{attribute 'c++_compatible'}
{attribute 'external_name' := 'EncoderTouchProbeRef_GUID_799525EC_5EF1_E852_EDA3_1BA0CDBD1FD9'}
{attribute 'TcIecLibraryType'}
{attribute 'no_explicit_call' :='do not call this POU directly'}
{attribute 'no_assign_warning'}
(* TouchProbeRef for Encoder Touch Probe. *)
FUNCTION_BLOCK EncoderTouchProbeRef
VAR
END_VAR
VAR_INPUT
	(* Settings for incremental encoder touch probe source selection. *)
	{attribute 'GUID' := '150DF3A8-F3D9-498D-A6F5-12073AD04A71'}
	{attribute 'Namespace' := 'Tc3_Mc3Ptp'}
	IncrementalEncoderSettings : IncrementalEncoderTouchProbeSettings;
END_VAR
VAR
	 {attribute 'hide'}
	_reserved1 : UDINT;
END_VAR
VAR_OUTPUT
	(* Connect to MC_TouchProbe/MC_AbortTrigger TriggerInput *)
	{attribute 'GUID' := 'CC3262A1-A7A1-46D3-802E-9117404E77E7'}
	{attribute 'Namespace' := 'Tc3_Mc3Ptp'}
	Trigger : TRIGGER_REF;
END_VAR
VAR
	 {attribute 'hide'}
	_reserved2 : ARRAY [1..8] OF USINT;
END_VAR

{attribute 'TcTypeSystem'}

(* Internal method *)
{attribute 'hide'}
METHOD FB_init : BOOL
VAR_INPUT
	(*  if TRUE, the retain variables are initialized (warm start / cold start) *)
	bInitRetains : BOOL;
	(*  if TRUE, the instance afterwards gets moved into the copy code (online change) *)
	bInCopyCode : BOOL;
END_VAR
END_METHOD

{attribute 'TcTypeSystem'}

(* Internal method *)
{attribute 'hide'}
METHOD FB_reinit : BOOL
END_METHOD

{attribute 'TcTypeSystem'}

(* Internal method *)
{attribute 'hide'}
METHOD FB_exit : BOOL
VAR_INPUT
	(*  if TRUE, the exit method is called for exiting an instance that is copied afterwards (online change). *)
	bInCopyCode : BOOL;
END_VAR
END_METHOD

END_FUNCTION_BLOCK

// TouchProbe/TimestampTouchProbeRef

{attribute 'c++_compatible'}
{attribute 'external_name' := 'TimestampTouchProbeRef_GUID_B6855340_6F16_E41B_E060_D5170EE631A7'}
{attribute 'TcIecLibraryType'}
{attribute 'no_explicit_call' :='do not call this POU directly'}
{attribute 'no_assign_warning'}
(* TouchProbeRef for Timestamp Touch Probes. *)
FUNCTION_BLOCK TimestampTouchProbeRef
VAR
END_VAR
VAR_INPUT
	(* Link to Axis Touch Probe Object -> Oid. *)
	{attribute 'GUID' := '18071995-0000-0000-0000-00000000000F'}
	Oid AT %I* : GLOBAL.OTCID;
END_VAR
VAR
	 {attribute 'hide'}
	_reserved1 : UDINT;
END_VAR
VAR_OUTPUT
	(* Connect to MC_Touchprobe/MC_AbortTrigger TriggerInput *)
	{attribute 'GUID' := 'CC3262A1-A7A1-46D3-802E-9117404E77E7'}
	{attribute 'Namespace' := 'Tc3_Mc3Ptp'}
	Trigger : TRIGGER_REF;
END_VAR

{attribute 'TcTypeSystem'}

(* Internal method *)
{attribute 'hide'}
METHOD FB_init : BOOL
VAR_INPUT
	(*  if TRUE, the retain variables are initialized (warm start / cold start) *)
	bInitRetains : BOOL;
	(*  if TRUE, the instance afterwards gets moved into the copy code (online change) *)
	bInCopyCode : BOOL;
END_VAR
END_METHOD

{attribute 'TcTypeSystem'}

(* Internal method *)
{attribute 'hide'}
METHOD FB_reinit : BOOL
END_METHOD

{attribute 'TcTypeSystem'}

(* Internal method *)
{attribute 'hide'}
METHOD FB_exit : BOOL
VAR_INPUT
	(*  if TRUE, the exit method is called for exiting an instance that is copied afterwards (online change). *)
	bInCopyCode : BOOL;
END_VAR
END_METHOD

END_FUNCTION_BLOCK

// TouchProbe/FixedStopTouchProbeRef

{attribute 'c++_compatible'}
{attribute 'external_name' := 'FixedStopTouchProbeRef_GUID_6C680BDF_D95B_EB97_DB3C_C590086A417A'}
{attribute 'TcIecLibraryType'}
{attribute 'no_explicit_call' :='do not call this POU directly'}
{attribute 'no_assign_warning'}
(* TouchProbeRef for Fixed Stop Detection. *)
FUNCTION_BLOCK FixedStopTouchProbeRef
VAR
END_VAR
VAR_INPUT
	(* Link to Axis Touch Probe Object -> Oid. *)
	{attribute 'GUID' := '18071995-0000-0000-0000-00000000000F'}
	Oid AT %I* : GLOBAL.OTCID;
END_VAR
VAR
	 {attribute 'hide'}
	_reserved1 : UDINT;
END_VAR
VAR_INPUT
	(* Settings for Fixed Stop Detection *)
	{attribute 'GUID' := 'CB5E9FDE-923C-4F7A-BCB2-279EC887599F'}
	{attribute 'Namespace' := 'Tc3_Mc3Ptp'}
	Settings : FixedStopTouchProbeSettings;
END_VAR
VAR_OUTPUT
	(* Connect to MC_Touchprobe/MC_AbortTrigger TriggerInput *)
	{attribute 'GUID' := 'CC3262A1-A7A1-46D3-802E-9117404E77E7'}
	{attribute 'Namespace' := 'Tc3_Mc3Ptp'}
	Trigger : TRIGGER_REF;
END_VAR

{attribute 'TcTypeSystem'}

(* Internal method *)
{attribute 'hide'}
METHOD FB_init : BOOL
VAR_INPUT
	(*  if TRUE, the retain variables are initialized (warm start / cold start) *)
	bInitRetains : BOOL;
	(*  if TRUE, the instance afterwards gets moved into the copy code (online change) *)
	bInCopyCode : BOOL;
END_VAR
END_METHOD

{attribute 'TcTypeSystem'}

(* Internal method *)
{attribute 'hide'}
METHOD FB_reinit : BOOL
END_METHOD

{attribute 'TcTypeSystem'}

(* Internal method *)
{attribute 'hide'}
METHOD FB_exit : BOOL
VAR_INPUT
	(*  if TRUE, the exit method is called for exiting an instance that is copied afterwards (online change). *)
	bInCopyCode : BOOL;
END_VAR
END_METHOD

END_FUNCTION_BLOCK

// Load Control/MC_LoadControl

{attribute 'c++_compatible'}
{attribute 'external_name' := 'MC_LoadControl_GUID_66886162_A3C4_E2E4_F654_8D3CE3C1FC4A'}
{attribute 'TcIecLibraryType'}
{attribute 'hide_all_locals'}
(* 
	This function block continuously exerts a torque, force or pressure of the specified value. <br/>
	Positive torque, force and differential pressure is in the positive direction of velocity, pressure is
	physically unsigned. LoadUnit must match the unit of the value measured by the corresponding sensor.
	 *)
FUNCTION_BLOCK MC_LoadControl
VAR_IN_OUT
	(* Reference to the axis *)
	{attribute 'GUID' := '931209B0-6FAC-E9BE-F824-23CE2FAA5732'}
	{attribute 'Namespace' := 'Tc3_Mc3Ptp'}
	Axis : AXIS_REF;
END_VAR
VAR_INPUT
	(* Start the motion at rising edge. *)
	Execute : BOOL;
END_VAR
VAR
	 {attribute 'hide'}
	_reserved1 : ARRAY [1..7] OF USINT;
END_VAR
VAR_INPUT
	(* Commanded load value ([LoadUnit]). It is approached using a defined ramp (LoadRamp). *)
	Load : LREAL := STRING_TO_LREAL('#Invalid');
	(* Maximum load derivative ([LoadUnit/s], positive) *)
	LoadRamp : LREAL := STRING_TO_LREAL('#Invalid');
	(* Maximum load ramp derivative ([LoadUnit/s^2], positive). It can be left as 'Ignore' if no ramp derivative limit is desired. *)
	LoadRampDerivative : LREAL := STRING_TO_LREAL('#Ignore');
	(* Chronological sequence of the command *)
	{attribute 'Namespace' := 'Tc3_Mc3Base'}
	BufferMode : Tc3_Mc3Base.EBufferMode := Tc3_Mc3Base.EBufferMode.Aborting;
END_VAR
VAR_OUTPUT
	(* Commanded load value reached *)
	InLoad : BOOL;
	(* Function block is not finished and new output values are to be expected. *)
	Busy : BOOL;
	(* Function block has active control on the axis. *)
	Active : BOOL;
	(* Command is aborted by another command. *)
	CommandAborted : BOOL;
	(* Error occurred within function block. *)
	Error : BOOL;
END_VAR
VAR
	 {attribute 'hide'}
	_reserved2 : USINT;
END_VAR
VAR_OUTPUT
	(* Error identifier *)
	ErrorId : UDINT;
END_VAR
VAR
	 {attribute 'hide'}
	_reserved3 : UINT_0_32;
	 {attribute 'hide'}
	_reserved4 : ARRAY [1..28] OF UINT_8_16;
	 {attribute 'hide'}
	_reserved5 : ARRAY [1..32] OF USINT;
END_VAR

{attribute 'TcTypeSystem'}

(* Internal method *)
{attribute 'hide'}
METHOD FB_init : BOOL
VAR_INPUT
	(*  if TRUE, the retain variables are initialized (warm start / cold start) *)
	bInitRetains : BOOL;
	(*  if TRUE, the instance afterwards gets moved into the copy code (online change) *)
	bInCopyCode : BOOL;
END_VAR
END_METHOD

{attribute 'TcTypeSystem'}

(* Internal method *)
{attribute 'hide'}
METHOD FB_exit : BOOL
VAR_INPUT
	(*  if TRUE, the exit method is called for exiting an instance that is copied afterwards (online change). *)
	bInCopyCode : BOOL;
END_VAR
END_METHOD

END_FUNCTION_BLOCK

// Administrative/Status/MC_ReadActualPosition

{attribute 'c++_compatible'}
{attribute 'external_name' := 'MC_ReadActualPosition_GUID_2E787536_22C6_ED03_C885_6ED50CC1B12A'}
{attribute 'TcIecLibraryType'}
{attribute 'hide_all_locals'}
(* 
		This function block reads the current axis actual position.<br/>
		In case of an invalid actual position value, the Position output is set to 0 and the Valid output is set to FALSE.
	 *)
FUNCTION_BLOCK MC_ReadActualPosition
VAR_IN_OUT
	(* Reference to the axis *)
	{attribute 'GUID' := '931209B0-6FAC-E9BE-F824-23CE2FAA5732'}
	{attribute 'Namespace' := 'Tc3_Mc3Ptp'}
	Axis : AXIS_REF;
END_VAR
VAR_INPUT
	(* Read the actual position continuously while Enable = TRUE. *)
	Enable : BOOL;
END_VAR
VAR_OUTPUT
	(* Valid output available at function block *)
	Valid : BOOL;
	(* Function block is not finished and new output values are to be expected. *)
	Busy : BOOL;
	(* Error occurred within function block. *)
	Error : BOOL;
	(* Error identifier *)
	ErrorId : UDINT;
	(* Actual position ([PosUnit]) *)
	Position : LREAL;
END_VAR

{attribute 'TcTypeSystem'}

(* Internal method *)
{attribute 'hide'}
METHOD FB_init : BOOL
VAR_INPUT
	(*  if TRUE, the retain variables are initialized (warm start / cold start) *)
	bInitRetains : BOOL;
	(*  if TRUE, the instance afterwards gets moved into the copy code (online change) *)
	bInCopyCode : BOOL;
END_VAR
END_METHOD

{attribute 'TcTypeSystem'}

(* Internal method *)
{attribute 'hide'}
METHOD FB_exit : BOOL
VAR_INPUT
	(*  if TRUE, the exit method is called for exiting an instance that is copied afterwards (online change). *)
	bInCopyCode : BOOL;
END_VAR
END_METHOD

END_FUNCTION_BLOCK

// Administrative/Status/MC_ReadActualTorque

{attribute 'c++_compatible'}
{attribute 'external_name' := 'MC_ReadActualTorque_GUID_AD684BB3_AFE8_E183_D73B_36C41C0C538D'}
{attribute 'TcIecLibraryType'}
{attribute 'hide_all_locals'}
(* 
		This function block reads the current axis actual torque.<br/>
		In case of an invalid actual torque value, the Torque output is set to 0 and the Valid output is set to FALSE.
	 *)
FUNCTION_BLOCK MC_ReadActualTorque
VAR_IN_OUT
	(* Reference to the axis *)
	{attribute 'GUID' := '931209B0-6FAC-E9BE-F824-23CE2FAA5732'}
	{attribute 'Namespace' := 'Tc3_Mc3Ptp'}
	Axis : AXIS_REF;
END_VAR
VAR_INPUT
	(* Read the actual torque continuously while Enable = TRUE. *)
	Enable : BOOL;
END_VAR
VAR_OUTPUT
	(* Valid output available at function block *)
	Valid : BOOL;
	(* Function block is not finished and new output values are to be expected. *)
	Busy : BOOL;
	(* Error occurred within function block. *)
	Error : BOOL;
	(* Error identifier *)
	ErrorId : UDINT;
	(* Actual torque ([TorqueUnit]) *)
	Torque : LREAL;
END_VAR

{attribute 'TcTypeSystem'}

(* Internal method *)
{attribute 'hide'}
METHOD FB_init : BOOL
VAR_INPUT
	(*  if TRUE, the retain variables are initialized (warm start / cold start) *)
	bInitRetains : BOOL;
	(*  if TRUE, the instance afterwards gets moved into the copy code (online change) *)
	bInCopyCode : BOOL;
END_VAR
END_METHOD

{attribute 'TcTypeSystem'}

(* Internal method *)
{attribute 'hide'}
METHOD FB_exit : BOOL
VAR_INPUT
	(*  if TRUE, the exit method is called for exiting an instance that is copied afterwards (online change). *)
	bInCopyCode : BOOL;
END_VAR
END_METHOD

END_FUNCTION_BLOCK

// Administrative/Status/MC_ReadActualVelocity

{attribute 'c++_compatible'}
{attribute 'external_name' := 'MC_ReadActualVelocity_GUID_DD1D8D4C_516C_E0E0_F57B_12AC9CA1B220'}
{attribute 'TcIecLibraryType'}
{attribute 'hide_all_locals'}
(* 
		This function block reads the current axis actual velocity.<br/>
		In case of an invalid actual velocity value, the Velocity output is set to 0 and the Valid output is set to FALSE.
	 *)
FUNCTION_BLOCK MC_ReadActualVelocity
VAR_IN_OUT
	(* Reference to the axis *)
	{attribute 'GUID' := '931209B0-6FAC-E9BE-F824-23CE2FAA5732'}
	{attribute 'Namespace' := 'Tc3_Mc3Ptp'}
	Axis : AXIS_REF;
END_VAR
VAR_INPUT
	(* Read the actual velocity continuously while Enable = TRUE. *)
	Enable : BOOL;
END_VAR
VAR_OUTPUT
	(* Valid output available at function block *)
	Valid : BOOL;
	(* Function block is not finished and new output values are to be expected. *)
	Busy : BOOL;
	(* Error occurred within function block. *)
	Error : BOOL;
	(* Error identifier *)
	ErrorId : UDINT;
	(* Actual velocity ([PosUnit]/s) *)
	Velocity : LREAL;
END_VAR

{attribute 'TcTypeSystem'}

(* Internal method *)
{attribute 'hide'}
METHOD FB_init : BOOL
VAR_INPUT
	(*  if TRUE, the retain variables are initialized (warm start / cold start) *)
	bInitRetains : BOOL;
	(*  if TRUE, the instance afterwards gets moved into the copy code (online change) *)
	bInCopyCode : BOOL;
END_VAR
END_METHOD

{attribute 'TcTypeSystem'}

(* Internal method *)
{attribute 'hide'}
METHOD FB_exit : BOOL
VAR_INPUT
	(*  if TRUE, the exit method is called for exiting an instance that is copied afterwards (online change). *)
	bInCopyCode : BOOL;
END_VAR
END_METHOD

END_FUNCTION_BLOCK

// Administrative/Status/MC_ReadAxisError

{attribute 'c++_compatible'}
{attribute 'external_name' := 'MC_ReadAxisError_GUID_161A2F0B_30EC_E528_DEE0_A4EC734D4B38'}
{attribute 'TcIecLibraryType'}
{attribute 'hide_all_locals'}
(* 
		This function block reads the current axis error identifier.
	 *)
FUNCTION_BLOCK MC_ReadAxisError
VAR_IN_OUT
	(* Reference to the axis *)
	{attribute 'GUID' := '931209B0-6FAC-E9BE-F824-23CE2FAA5732'}
	{attribute 'Namespace' := 'Tc3_Mc3Ptp'}
	Axis : AXIS_REF;
END_VAR
VAR_INPUT
	(* Read the axis error identifier continuously while Enable = TRUE. *)
	Enable : BOOL;
END_VAR
VAR_OUTPUT
	(* Valid output available at function block *)
	Valid : BOOL;
	(* Function block is not finished and new output values are to be expected. *)
	Busy : BOOL;
	(* Error occurred within function block. *)
	Error : BOOL;
	(* Error identifier *)
	ErrorId : UDINT;
	(* Axis error identifier *)
	AxisErrorId : UDINT;
END_VAR
VAR
	 {attribute 'hide'}
	_reserved1 : UINT_0_32;
END_VAR

{attribute 'TcTypeSystem'}

(* Internal method *)
{attribute 'hide'}
METHOD FB_init : BOOL
VAR_INPUT
	(*  if TRUE, the retain variables are initialized (warm start / cold start) *)
	bInitRetains : BOOL;
	(*  if TRUE, the instance afterwards gets moved into the copy code (online change) *)
	bInCopyCode : BOOL;
END_VAR
END_METHOD

{attribute 'TcTypeSystem'}

(* Internal method *)
{attribute 'hide'}
METHOD FB_exit : BOOL
VAR_INPUT
	(*  if TRUE, the exit method is called for exiting an instance that is copied afterwards (online change). *)
	bInCopyCode : BOOL;
END_VAR
END_METHOD

END_FUNCTION_BLOCK

// Administrative/Status/MC_ReadStatus

{attribute 'c++_compatible'}
{attribute 'external_name' := 'MC_ReadStatus_GUID_BDF6D356_383A_E775_CF5E_17BC66992CB4'}
{attribute 'TcIecLibraryType'}
{attribute 'hide_all_locals'}
(* 
		This function block reads the current axis state.
	 *)
FUNCTION_BLOCK MC_ReadStatus
VAR_IN_OUT
	(* Reference to the axis *)
	{attribute 'GUID' := '931209B0-6FAC-E9BE-F824-23CE2FAA5732'}
	{attribute 'Namespace' := 'Tc3_Mc3Ptp'}
	Axis : AXIS_REF;
END_VAR
VAR_INPUT
	(* Read the axis state continuously while Enable = TRUE. *)
	Enable : BOOL;
END_VAR
VAR_OUTPUT
	(* Valid output available at function block *)
	Valid : BOOL;
	(* Function block is not finished and new output values are to be expected. *)
	Busy : BOOL;
	(* Error occurred within function block. *)
	Error : BOOL;
	(* Error identifier *)
	ErrorId : UDINT;
	(* Axis is in state ErrorStop. *)
	ErrorStop : BOOL;
	(* Axis is in state Disabled. *)
	Disabled : BOOL;
	(* Axis is in state Stopping. *)
	Stopping : BOOL;
	(* Axis is in state Homing. *)
	Homing : BOOL;
	(* Axis is in state Standstill. *)
	Standstill : BOOL;
	(* Axis is in state DiscreteMotion. *)
	DiscreteMotion : BOOL;
	(* Axis is in state ContinuousMotion. *)
	ContinuousMotion : BOOL;
	(* Axis is in state SynchronizedMotion. *)
	SynchronizedMotion : BOOL;
END_VAR

{attribute 'TcTypeSystem'}

(* Internal method *)
{attribute 'hide'}
METHOD FB_init : BOOL
VAR_INPUT
	(*  if TRUE, the retain variables are initialized (warm start / cold start) *)
	bInitRetains : BOOL;
	(*  if TRUE, the instance afterwards gets moved into the copy code (online change) *)
	bInCopyCode : BOOL;
END_VAR
END_METHOD

{attribute 'TcTypeSystem'}

(* Internal method *)
{attribute 'hide'}
METHOD FB_exit : BOOL
VAR_INPUT
	(*  if TRUE, the exit method is called for exiting an instance that is copied afterwards (online change). *)
	bInCopyCode : BOOL;
END_VAR
END_METHOD

END_FUNCTION_BLOCK

// Administrative/Parameter/MC_WriteHardwareParameter

{attribute 'c++_compatible'}
{attribute 'external_name' := 'MC_WriteHardwareParameter_GUID_4D6A3EB3_2727_E24A_E1EB_F69B71611CB4'}
{attribute 'TcIecLibraryType'}
{attribute 'hide_all_locals'}
(* 
		This function block allows to write parameters to the hardware drive asynchronously via ADS. It supports CoE and SoE drives.
	 *)
FUNCTION_BLOCK MC_WriteHardwareParameter
VAR_IN_OUT
	(* Reference to the axis *)
	{attribute 'GUID' := '931209B0-6FAC-E9BE-F824-23CE2FAA5732'}
	{attribute 'Namespace' := 'Tc3_Mc3Ptp'}
	Axis : AXIS_REF;
END_VAR
VAR_INPUT
	(* Rising edge triggers the write operation. *)
	Execute : BOOL;
END_VAR
VAR
	 {attribute 'hide'}
	_reserved1 : USINT;
END_VAR
VAR_INPUT
	(* CoE object index or SoE IDN *)
	Index : UINT := 0;
	(* CoE sub index or SoE element *)
	SubIndex : USINT := 0;
END_VAR
VAR
	 {attribute 'hide'}
	_reserved2 : ARRAY [1..3] OF USINT;
END_VAR
VAR_INPUT
	(* Contains the address of the data. *)
	{attribute 'GUID' := '18071995-0000-0000-0000-000000000018'}
	SourceAddress : GLOBAL.PVOID := 0;
	(* Contains the size of the data. *)
	DataSize : UDINT := 0;
END_VAR
VAR_OUTPUT
	(* Value is successfully sent to the target. *)
	Done : BOOL;
	(* Function block is not finished. *)
	Busy : BOOL;
	(* Function block is active. *)
	Active : BOOL;
	(* Error occurred within function block. *)
	Error : BOOL;
	(* Error identifier *)
	ErrorId : UDINT;
END_VAR
VAR
	 {attribute 'hide'}
	_reserved3 : UINT_0_32;
	 {attribute 'hide'}
	_reserved4 : ARRAY [1..32] OF UINT_8_16;
	 {attribute 'hide'}
	_reserved5 : ARRAY [1..32] OF USINT;
END_VAR

{attribute 'TcTypeSystem'}

(* Internal method *)
{attribute 'hide'}
METHOD FB_init : BOOL
VAR_INPUT
	(*  if TRUE, the retain variables are initialized (warm start / cold start) *)
	bInitRetains : BOOL;
	(*  if TRUE, the instance afterwards gets moved into the copy code (online change) *)
	bInCopyCode : BOOL;
END_VAR
END_METHOD

{attribute 'TcTypeSystem'}

(* Internal method *)
{attribute 'hide'}
METHOD FB_exit : BOOL
VAR_INPUT
	(*  if TRUE, the exit method is called for exiting an instance that is copied afterwards (online change). *)
	bInCopyCode : BOOL;
END_VAR
END_METHOD

END_FUNCTION_BLOCK

// Administrative/Parameter/MC_ReadHardwareParameter

{attribute 'c++_compatible'}
{attribute 'external_name' := 'MC_ReadHardwareParameter_GUID_DBC0D23F_EDB5_E904_FCD0_3F6DCE5C9980'}
{attribute 'TcIecLibraryType'}
{attribute 'hide_all_locals'}
(* 
		This function block allows to read parameters from the hardware drive asynchronously via ADS. The function block supports CoE and SoE drives.
	 *)
FUNCTION_BLOCK MC_ReadHardwareParameter
VAR_IN_OUT
	(* Reference to the axis *)
	{attribute 'GUID' := '931209B0-6FAC-E9BE-F824-23CE2FAA5732'}
	{attribute 'Namespace' := 'Tc3_Mc3Ptp'}
	Axis : AXIS_REF;
END_VAR
VAR_INPUT
	(* Trigger the command with rising edge. *)
	Execute : BOOL;
END_VAR
VAR
	 {attribute 'hide'}
	_reserved1 : USINT;
END_VAR
VAR_INPUT
	(* CoE object index or SoE IDN *)
	Index : UINT := 0;
	(* CoE sub index or SoE element *)
	SubIndex : USINT := 0;
END_VAR
VAR
	 {attribute 'hide'}
	_reserved2 : ARRAY [1..3] OF USINT;
END_VAR
VAR_INPUT
	(* Contains the address of the destination buffer. *)
	{attribute 'GUID' := '18071995-0000-0000-0000-000000000018'}
	DestinationAddress : GLOBAL.PVOID := 0;
	(* Contains the size of the destination buffer. *)
	DataSize : UDINT := 0;
END_VAR
VAR_OUTPUT
	(* Value is successfully read from the target. *)
	Done : BOOL;
	(* Function block is not finished. *)
	Busy : BOOL;
	(* Function block is active. *)
	Active : BOOL;
	(* Error occurred within function block. *)
	Error : BOOL;
	(* Error identifier *)
	ErrorId : UDINT;
END_VAR
VAR
	 {attribute 'hide'}
	_reserved3 : UINT_0_32;
	 {attribute 'hide'}
	_reserved4 : ARRAY [1..32] OF UINT_8_16;
	 {attribute 'hide'}
	_reserved5 : ARRAY [1..32] OF USINT;
END_VAR

{attribute 'TcTypeSystem'}

(* Internal method *)
{attribute 'hide'}
METHOD FB_init : BOOL
VAR_INPUT
	(*  if TRUE, the retain variables are initialized (warm start / cold start) *)
	bInitRetains : BOOL;
	(*  if TRUE, the instance afterwards gets moved into the copy code (online change) *)
	bInCopyCode : BOOL;
END_VAR
END_METHOD

{attribute 'TcTypeSystem'}

(* Internal method *)
{attribute 'hide'}
METHOD FB_exit : BOOL
VAR_INPUT
	(*  if TRUE, the exit method is called for exiting an instance that is copied afterwards (online change). *)
	bInCopyCode : BOOL;
END_VAR
END_METHOD

END_FUNCTION_BLOCK

// Administrative/Parameter/MC_ReadParameter

{attribute 'c++_compatible'}
{attribute 'pack_mode' := '1'}
{attribute 'external_name' := 'MC_ReadParameter_GUID_FFD552A7_9EB3_EE4D_D310_ABB0C47D1F25'}
{attribute 'TcIecLibraryType'}
{attribute 'hide_all_locals'}
(* 
		This function block reads a numeric (LREAL) parameter value from the axis.<br/>
		The command is typically processed synchronously.
	 *)
FUNCTION_BLOCK MC_ReadParameter
VAR_INPUT
	(* Reference to the axis *)
	{attribute 'GUID' := 'BAA3CD7D-9477-45D8-9B5E-5D0F462A0EBD'}
	{attribute 'Namespace' := 'Tc3_Mc3Ptp'}
	Axis : Type_PtpReadWriteParameter;
	(* Triggers a read on rising edge (EReadMode.Once) or every cycle while TRUE (EReadMode.Cyclic). *)
	Enable : BOOL;
END_VAR
VAR
	 {attribute 'hide'}
	_reserved1 : UINT_24_56;
END_VAR
VAR_INPUT
	(* Identifier of the parameter to read. *)
	{attribute 'GUID' := 'C0077006-E40F-45AC-AC09-497A34D67EFE'}
	{attribute 'Namespace' := 'Tc3_Mc3Ptp'}
	ParameterId : EAxisParameterId := EAxisParameterId.Invalid;
	(* Once: read once at rising edge of Enable. Cyclic: read every cycle while Enable is TRUE. *)
	{attribute 'GUID' := '0E6410AA-E380-4C0B-A4DF-BBE8E3558B02'}
	{attribute 'Namespace' := 'Tc3_Mc3Ptp'}
	Mode : EReadMode := EReadMode.Once;
END_VAR
VAR_OUTPUT
	(* Valid output available at function block. *)
	Valid : BOOL;
	(* Function block is not finished. Always FALSE with ReadMode Once. *)
	Busy : BOOL;
	(* Error occurred within function block. *)
	Error : BOOL;
END_VAR
VAR
	 {attribute 'hide'}
	_reserved2 : USINT;
END_VAR
VAR_OUTPUT
	(* Error identifier *)
	ErrorId : UDINT;
END_VAR
VAR
	 {attribute 'hide'}
	_reserved3 : UDINT;
END_VAR
VAR_OUTPUT
	(* Last successfully read value of the parameter. *)
	Value : LREAL;
END_VAR
VAR
	 {attribute 'hide'}
	_reserved4 : ARRAY [1..8] OF USINT;
END_VAR

{attribute 'TcTypeSystem'}

(* Internal method *)
{attribute 'hide'}
METHOD FB_init : BOOL
VAR_INPUT
	(*  if TRUE, the retain variables are initialized (warm start / cold start) *)
	bInitRetains : BOOL;
	(*  if TRUE, the instance afterwards gets moved into the copy code (online change) *)
	bInCopyCode : BOOL;
END_VAR
END_METHOD

{attribute 'TcTypeSystem'}

(* Internal method *)
{attribute 'hide'}
METHOD FB_exit : BOOL
VAR_INPUT
	(*  if TRUE, the exit method is called for exiting an instance that is copied afterwards (online change). *)
	bInCopyCode : BOOL;
END_VAR
END_METHOD

END_FUNCTION_BLOCK

// Administrative/Parameter/MC_WriteParameter

{attribute 'c++_compatible'}
{attribute 'pack_mode' := '1'}
{attribute 'external_name' := 'MC_WriteParameter_GUID_E0C44196_E982_ED5C_E203_9AA7356E2026'}
{attribute 'TcIecLibraryType'}
{attribute 'hide_all_locals'}
(* 
		This function block writes a numeric (LREAL) parameter value to the axis.<br/>
		The command is typically processed synchronously.
	 *)
FUNCTION_BLOCK MC_WriteParameter
VAR_INPUT
	(* Reference to the axis *)
	{attribute 'GUID' := 'BAA3CD7D-9477-45D8-9B5E-5D0F462A0EBD'}
	{attribute 'Namespace' := 'Tc3_Mc3Ptp'}
	Axis : Type_PtpReadWriteParameter;
	(* Trigger the command with rising edge. *)
	Execute : BOOL;
END_VAR
VAR
	 {attribute 'hide'}
	_reserved1 : UINT_24_56;
END_VAR
VAR_INPUT
	(* Identifier of the parameter to write. *)
	{attribute 'GUID' := 'C0077006-E40F-45AC-AC09-497A34D67EFE'}
	{attribute 'Namespace' := 'Tc3_Mc3Ptp'}
	ParameterId : EAxisParameterId := EAxisParameterId.Invalid;
	(* Value of the parameter to write. *)
	Value : LREAL;
END_VAR
VAR_OUTPUT
	(* Parameter value has been successfully written. *)
	Done : BOOL;
	(* Function block is not finished. *)
	Busy : BOOL;
	(* Error occurred within function block. *)
	Error : BOOL;
END_VAR
VAR
	 {attribute 'hide'}
	_reserved2 : USINT;
END_VAR
VAR_OUTPUT
	(* Error identifier *)
	ErrorId : UDINT;
END_VAR
VAR
	 {attribute 'hide'}
	_reserved3 : ARRAY [1..8] OF USINT;
END_VAR

{attribute 'TcTypeSystem'}

(* Internal method *)
{attribute 'hide'}
METHOD FB_init : BOOL
VAR_INPUT
	(*  if TRUE, the retain variables are initialized (warm start / cold start) *)
	bInitRetains : BOOL;
	(*  if TRUE, the instance afterwards gets moved into the copy code (online change) *)
	bInCopyCode : BOOL;
END_VAR
END_METHOD

{attribute 'TcTypeSystem'}

(* Internal method *)
{attribute 'hide'}
METHOD FB_exit : BOOL
VAR_INPUT
	(*  if TRUE, the exit method is called for exiting an instance that is copied afterwards (online change). *)
	bInCopyCode : BOOL;
END_VAR
END_METHOD

END_FUNCTION_BLOCK

// Administrative/Parameter/MC_ReadBoolParameter

{attribute 'c++_compatible'}
{attribute 'pack_mode' := '1'}
{attribute 'external_name' := 'MC_ReadBoolParameter_GUID_CEBA038E_F895_EC6F_FD72_8D56265F8337'}
{attribute 'TcIecLibraryType'}
{attribute 'hide_all_locals'}
(* 
		This function block reads a boolean parameter value from the axis.<br/>
		The command is typically processed synchronously.
	 *)
FUNCTION_BLOCK MC_ReadBoolParameter
VAR_INPUT
	(* Reference to the axis *)
	{attribute 'GUID' := 'BAA3CD7D-9477-45D8-9B5E-5D0F462A0EBD'}
	{attribute 'Namespace' := 'Tc3_Mc3Ptp'}
	Axis : Type_PtpReadWriteParameter;
	(* Triggers a read on rising edge (EReadMode.Once) or every cycle while TRUE (EReadMode.Cyclic). *)
	Enable : BOOL;
END_VAR
VAR
	 {attribute 'hide'}
	_reserved1 : UINT_24_56;
END_VAR
VAR_INPUT
	(* Identifier of the parameter to read. *)
	{attribute 'GUID' := 'C0077006-E40F-45AC-AC09-497A34D67EFE'}
	{attribute 'Namespace' := 'Tc3_Mc3Ptp'}
	ParameterId : EAxisParameterId := EAxisParameterId.Invalid;
	(* Once: read once at rising edge of Enable. Cyclic: read every cycle while Enable is TRUE. *)
	{attribute 'GUID' := '0E6410AA-E380-4C0B-A4DF-BBE8E3558B02'}
	{attribute 'Namespace' := 'Tc3_Mc3Ptp'}
	Mode : EReadMode := EReadMode.Once;
END_VAR
VAR_OUTPUT
	(* Valid output available at function block. *)
	Valid : BOOL;
	(* Function block is not finished. Always FALSE with ReadMode Once. *)
	Busy : BOOL;
	(* Error occurred within function block. *)
	Error : BOOL;
END_VAR
VAR
	 {attribute 'hide'}
	_reserved2 : USINT;
END_VAR
VAR_OUTPUT
	(* Error identifier *)
	ErrorId : UDINT;
	(* Last successfully read value of the parameter. *)
	Value : BOOL;
END_VAR
VAR
	 {attribute 'hide'}
	_reserved3 : ARRAY [1..3] OF USINT;
END_VAR

{attribute 'TcTypeSystem'}

(* Internal method *)
{attribute 'hide'}
METHOD FB_init : BOOL
VAR_INPUT
	(*  if TRUE, the retain variables are initialized (warm start / cold start) *)
	bInitRetains : BOOL;
	(*  if TRUE, the instance afterwards gets moved into the copy code (online change) *)
	bInCopyCode : BOOL;
END_VAR
END_METHOD

{attribute 'TcTypeSystem'}

(* Internal method *)
{attribute 'hide'}
METHOD FB_exit : BOOL
VAR_INPUT
	(*  if TRUE, the exit method is called for exiting an instance that is copied afterwards (online change). *)
	bInCopyCode : BOOL;
END_VAR
END_METHOD

END_FUNCTION_BLOCK

// Administrative/Parameter/MC_WriteBoolParameter

{attribute 'c++_compatible'}
{attribute 'pack_mode' := '1'}
{attribute 'external_name' := 'MC_WriteBoolParameter_GUID_DDAB129F_CB64_E37E_EC65_7C4517409200'}
{attribute 'TcIecLibraryType'}
{attribute 'hide_all_locals'}
(* 
		This function block writes a boolean parameter value to the axis.<br/>
		The command is typically processed synchronously.
	 *)
FUNCTION_BLOCK MC_WriteBoolParameter
VAR_INPUT
	(* Reference to the axis *)
	{attribute 'GUID' := 'BAA3CD7D-9477-45D8-9B5E-5D0F462A0EBD'}
	{attribute 'Namespace' := 'Tc3_Mc3Ptp'}
	Axis : Type_PtpReadWriteParameter;
	(* Trigger the command with rising edge. *)
	Execute : BOOL;
END_VAR
VAR
	 {attribute 'hide'}
	_reserved1 : UINT_24_56;
END_VAR
VAR_INPUT
	(* Identifier of the parameter to write. *)
	{attribute 'GUID' := 'C0077006-E40F-45AC-AC09-497A34D67EFE'}
	{attribute 'Namespace' := 'Tc3_Mc3Ptp'}
	ParameterId : EAxisParameterId := EAxisParameterId.Invalid;
	(* Value of the parameter to write. *)
	Value : BOOL;
END_VAR
VAR_OUTPUT
	(* Parameter value has been successfully written. *)
	Done : BOOL;
	(* Function block is not finished. *)
	Busy : BOOL;
	(* Error occurred within function block. *)
	Error : BOOL;
	(* Error identifier *)
	ErrorId : UDINT;
END_VAR
VAR
	 {attribute 'hide'}
	_reserved2 : ARRAY [1..4] OF UINT_8_16;
END_VAR

{attribute 'TcTypeSystem'}

(* Internal method *)
{attribute 'hide'}
METHOD FB_init : BOOL
VAR_INPUT
	(*  if TRUE, the retain variables are initialized (warm start / cold start) *)
	bInitRetains : BOOL;
	(*  if TRUE, the instance afterwards gets moved into the copy code (online change) *)
	bInCopyCode : BOOL;
END_VAR
END_METHOD

{attribute 'TcTypeSystem'}

(* Internal method *)
{attribute 'hide'}
METHOD FB_exit : BOOL
VAR_INPUT
	(*  if TRUE, the exit method is called for exiting an instance that is copied afterwards (online change). *)
	bInCopyCode : BOOL;
END_VAR
END_METHOD

END_FUNCTION_BLOCK
